FUNCTION_BLOCK ABSTRACT FB_AxisBase EXTENDS FB_ComponentBase IMPLEMENTS ITF_AxisBase
VAR CONSTANT
	//Constant declarations
	AXIS_BASE_ALARM_COUNT	: UDINT := 16;
END_VAR

VAR
	//ITF_AxisBase internal property variables
	fJogFastVelocity	: LREAL;
	fJogSlowVelocity	: LREAL;
	fTargetVelocity		: LREAL;
	
	bDriveEnabled		: BOOL;
	bInGear				: BOOL;
	bInPosition			: BOOL;
	fPosition 			: LREAL;
	fPositionSetpoint	: LREAL;
	bStopped			: BOOL;
	
	//Axis MC function blocks
	fbAxisJog: MC_Jog;
	fbAxisPower: MC_Power;
	fbAxisReset: MC_Reset;
	fbMoveAbsolute: MC_MoveAbsolute;
	fbMoveVelocity: MC_MoveVelocity;
	fbMoveRelative: MC_MoveRelative;
	fbAxisHalt: MC_Halt;
	fbAxisStop: MC_Stop;
	fbAxisHome: MC_Home;
	fbGearIn: MC_GearIn;
	fbResetDrv: FB_SoEReset;
	fbWriteParameter : MC_WriteParameter;
	
	//Alarming
	fbAxisBaseAlarms : ARRAY[1..AXIS_BASE_ALARM_COUNT] OF FB_TcAlarm;
	
	//Internal Variables
	fOverride		: LREAL := 100;		//Velocity Override
	SelectedAxis	: REFERENCE TO AXIS_REF REF= SimulationAxis;	//TODO: Make a better simulation system
	SimulationAxis: AXIS_REF;
	HardwareAxis: AXIS_REF;

	sTemp: STRING;
	stAxisBaseHMI		: ST_AxisBase_HMI;
	
	nAxisCopy: INT;
	bParamCopyComplete: BOOL;
END_VAR
VAR_IN_OUT
	MasterAxis	: AXIS_REF;
END_VAR

PROPERTY AxisRef : AXIS_REF
GET
AxisRef := SelectedAxis;
END_GET
END_PROPERTY

PROPERTY DriveEnabled : BOOL
GET
Enabled := bDriveEnabled;
END_GET
END_PROPERTY

METHOD ErrorOperation : BOOL
VAR_INPUT
END_VAR
SUPER^.ErrorOperation();

bEnabled := FALSE;
END_METHOD

METHOD GearInBasic : BOOL
VAR_IN_OUT
	master : AXIS_REF;	//Master axis to which the gearing will be made
END_VAR
IF NOT bActive THEN
	
	MasterAxis := master;		//"Master" must be specified in the FB call, so this particular variable is declared in the main FB and assigned from here
	fbGearIn.Execute := TRUE;
	
END_IF
END_METHOD

METHOD HardwareUpdate : BOOL
VAR_INPUT
END_VAR
SUPER^.HardwareUpdate();
	
//Resets the axis Drive Hardware when commanded by a "ResetDrive" Method call
fbResetDrv(
	NetId:= '', 
	Timeout:= T#10S, 
	Axis:= HardwareAxis);
	
fbResetDrv.Execute := FALSE;
END_METHOD

METHOD HMICommunication : BOOL
//Extend this method in extended FBs to communicate specific implementation data
SUPER^.HMICommunication();

//Process HMI requests
IF stAxisBaseHMI.bIncomingHMIRequest AND NOT stAxisBaseHMI.bHMICommandConfirmation THEN		//If a request has been issued by the HMI, and a previous request has not just finished being processed
	IF stAxisBaseHMI.bHMIControlAvailable THEN		//If the current conditions permit HMI control (Should be determined by the extended application components)
		IF stAxisBaseHMI.bDriveEnableHMIRequest THEN
			bEnabled := TRUE;
			stAxisBaseHMI.bHMICommandConfirmation := TRUE;	//Confirm that the request has been processed
		END_IF
		IF stAxisBaseHMI.bDriveDisableHMIRequest THEN
			bEnabled := FALSE;
			stAxisBaseHMI.bHMICommandConfirmation := TRUE;	//Confirm that the request has been processed
		END_IF
		IF stAxisBaseHMI.bSetJogFastVelocityRequest THEN
			fJogFastVelocity := stAxisBaseHMI.fSetJogFastVelocityValue;
			stAxisBaseHMI.bHMICommandConfirmation := TRUE;	//Confirm that the request has been processed
		END_IF
		IF stAxisBaseHMI.bSetJogSlowVelocityRequest THEN
			fJogSlowVelocity := stAxisBaseHMI.fSetJogSlowVelocityValue;
			stAxisBaseHMI.bHMICommandConfirmation := TRUE;	//Confirm that the request has been processed
		END_IF
		IF stAxisBaseHMI.bSetTargetVelocityRequest THEN
			fTargetVelocity := stAxisBaseHMI.bSetTargetVelocityValue;
			stAxisBaseHMI.bHMICommandConfirmation := TRUE;	//Confirm that the request has been processed
		END_IF
	END_IF
END_IF

//Update HMI status info
stAxisBaseHMI.fJogFastVelocity := fJogFastVelocity;
stAxisBaseHMI.fJogSlowVelocity := fJogSlowVelocity;
stAxisBaseHMI.fTargetVelocity := fTargetVelocity;
stAxisBaseHMI.bDriveEnabled := bDriveEnabled;
stAxisBaseHMI.bInGear := bInGear;
stAxisBaseHMI.bInPosition := bInPosition;
stAxisBaseHMI.fPosition := fPosition;
stAxisBaseHMI.fPositionSetpoint := fPositionSetpoint;
stAxisBaseHMI.bStopped := bStopped;
END_METHOD

METHOD Home : BOOL
//This method should be overridden by the extending FB based on the specific hardware configuration
END_METHOD

PROPERTY InGear : BOOL
GET
InGear := bInGear;
END_GET
END_PROPERTY

METHOD Inhibit : BOOL
VAR_INPUT
END_VAR
fbAxisPower.Override := 0;
END_METHOD

METHOD initialize : BOOL
VAR_INPUT
END_VAR

VAR
	sTemp: STRING;
END_VAR
SUPER^.initialize();

sTemp := CONCAT(CONCAT(CONCAT('Axis ', ': '), sName), ' '); 	//Creates a utility string for alarms and other messaging that reads (example text) - "Module 10 - Main Casepacker" to be followed by the alarm or message info
//TODO: Rename Event Class to AxisBase
F_CreateAllEventsInClass(	p_aAlarms := fbAxisBaseAlarms,
							nClassSize := SIZEOF(TC_EVENTS.AxisBase),
							pInitEvent := ADR(TC_EVENTS.AxisBase.InitReferenceEvent),
							sPrefix := sTemp );
END_METHOD

PROPERTY InPosition : BOOL
GET
InPosition := bInPosition;
END_GET
END_PROPERTY

METHOD Jog : BOOL
VAR_INPUT
	direction	: BOOL;			//"TRUE" for positive jog, "FALSE" for negative jog
	fast		: BOOL;			//"TRUE" for 'fast' jog, "FALSE" for 'slow' jog (As defined by Jog(Slow/Fast)Velocity Property)
END_VAR
//If the jog is currently active, allow the method to run again to ensure that the corresponding Jog bit can remain high so the jog can continue
//Otherwise, only start a jog when the axis is not already busy
IF fbAxisJog.Busy OR NOT bActive THEN
	
	fbAxisJog.JogForward:= direction; 
	fbAxisJog.JogBackwards:= NOT direction;
	
	IF fast THEN
		fbAxisJog.Velocity := fJogFastVelocity;
	ELSE
		fbAxisJog.Velocity := fJogSlowVelocity;
	END_IF
	
END_IF
END_METHOD

PROPERTY JogFastVelocity : LREAL
GET
JogFastVelocity : fJogFastVelocity;
END_GET
SET
fJogFastVelocity := JogFastVelocity;
END_SET
END_PROPERTY

PROPERTY JogSlowVelocity : LREAL
GET
JogSlowVelocity : fJogSlowVelocity;
END_GET
SET
fJogSlowVelocity : JogSlowVelocity;
END_SET
END_PROPERTY

METHOD Monitoring : BOOL
SUPER^.Monitoring();

//Cyclically updates the "Status" values from the NC-axis to the PLC (Axis1.Status...)
SelectedAxis.ReadStatus();

//Cyclically monitor all FB "Busy" bits, as well as the axis "HasJob" bit to ensure ADS communication time does not result in a delay before the "Busy" property is accurate after calling a FB
bActive := 		SimulationAxis.Status.HasJob
				OR	fbAxisJog.Busy
				OR	fbMoveAbsolute.Busy
				OR	fbMoveVelocity.Busy
				OR	fbMoveRelative.Busy
				OR	fbAxisHalt.Busy
				OR	fbAxisStop.Busy
				OR	fbAxisHome.Busy
				OR	fbGearIn.Busy;
				

//Update all internal property variables
bDriveEnabled := fbAxisPower.Status;
bInGear	:= (SelectedAxis.NcToPlc.CoupleState = 3);	//Note that this only looks for a simple gearing arrangement where this axis is a slave and not a master to any other axis
bInPosition := SelectedAxis.Status.InTargetPosition;
fPosition := SelectedAxis.NcToPlc.ActPos;
fPositionSetpoint := SelectedAxis.NcToPlc.SetPos;
bStopped := SelectedAxis.Status.StandStill;

				
//Error monitoring and event logging

IF fbAxisJog.Error AND NOT fbAxisBaseAlarms[E_AxisBase.JogError].bRaised THEN
	bError := TRUE;
	nErrorID := E_AxisBase.JogError;
	sTemp := UDINT_TO_STRING(fbAxisJog.ErrorID);
	fbAxisBaseAlarms[E_AxisBase.JogError].ipArguments.Clear().AddString(sName).AddString(sTemp);
	fbAxisBaseAlarms[E_AxisBase.JogError].Raise(0);
ELSIF NOT fbAxisJog.Error AND fbAxisBaseAlarms[E_AxisBase.JogError].bRaised THEN
	fbAxisBaseAlarms[E_AxisBase.JogError].Clear(0,0);
END_IF


IF fbAxisPower.Error AND NOT fbAxisBaseAlarms[E_AxisBase.PowerError].bRaised THEN
	bError := TRUE;
	nErrorID := E_AxisBase.PowerError;
	sTemp := UDINT_TO_STRING(fbAxisPower.ErrorID);
	fbAxisBaseAlarms[E_AxisBase.PowerError].ipArguments.Clear().AddString(sName).AddString(sTemp);
	fbAxisBaseAlarms[E_AxisBase.PowerError].Raise(0);
ELSIF NOT fbAxisPower.Error AND fbAxisBaseAlarms[E_AxisBase.PowerError].bRaised THEN
	fbAxisBaseAlarms[E_AxisBase.PowerError].Clear(0,0);
END_IF


IF fbAxisReset.Error AND NOT fbAxisBaseAlarms[E_AxisBase.ResetError].bRaised THEN
	bError := TRUE;
	nErrorID := E_AxisBase.ResetError;
	sTemp := UDINT_TO_STRING(fbAxisReset.ErrorID);
	fbAxisBaseAlarms[E_AxisBase.ResetError].ipArguments.Clear().AddString(sName).AddString(sTemp);
	fbAxisBaseAlarms[E_AxisBase.ResetError].Raise(0);
ELSIF NOT fbAxisReset.Error AND fbAxisBaseAlarms[E_AxisBase.ResetError].bRaised THEN
	fbAxisBaseAlarms[E_AxisBase.ResetError].Clear(0,0);
END_IF


IF fbMoveAbsolute.Error AND NOT fbAxisBaseAlarms[E_AxisBase.MoveAbsoluteError].bRaised THEN
	bError := TRUE;
	nErrorID := E_AxisBase.MoveAbsoluteError;
	sTemp := UDINT_TO_STRING(fbMoveAbsolute.ErrorID);
	fbAxisBaseAlarms[E_AxisBase.MoveAbsoluteError].ipArguments.Clear().AddString(sName).AddString(sTemp);
	fbAxisBaseAlarms[E_AxisBase.MoveAbsoluteError].Raise(0);
ELSIF NOT fbMoveAbsolute.Error AND fbAxisBaseAlarms[E_AxisBase.MoveAbsoluteError].bRaised THEN
	fbAxisBaseAlarms[E_AxisBase.MoveAbsoluteError].Clear(0,0);
END_IF


IF fbMoveVelocity.Error AND NOT fbAxisBaseAlarms[E_AxisBase.MoveVelocityError].bRaised THEN
	bError := TRUE;
	nErrorID := E_AxisBase.MoveVelocityError;
	sTemp := UDINT_TO_STRING(fbMoveVelocity.ErrorID);
	fbAxisBaseAlarms[E_AxisBase.MoveVelocityError].ipArguments.Clear().AddString(sName).AddString(sTemp);
	fbAxisBaseAlarms[E_AxisBase.MoveVelocityError].Raise(0);
ELSIF NOT fbMoveVelocity.Error AND fbAxisBaseAlarms[E_AxisBase.MoveVelocityError].bRaised THEN
	fbAxisBaseAlarms[E_AxisBase.MoveVelocityError].Clear(0,0);
END_IF


IF fbMoveRelative.Error AND NOT fbAxisBaseAlarms[E_AxisBase.MoveRelativeError].bRaised THEN
	bError := TRUE;
	nErrorID := E_AxisBase.MoveRelativeError;
	sTemp := UDINT_TO_STRING(fbMoveRelative.ErrorID);
	fbAxisBaseAlarms[E_AxisBase.MoveRelativeError].ipArguments.Clear().AddString(sName).AddString(sTemp);
	fbAxisBaseAlarms[E_AxisBase.MoveRelativeError].Raise(0);
ELSIF NOT fbMoveRelative.Error AND fbAxisBaseAlarms[E_AxisBase.MoveRelativeError].bRaised THEN
	fbAxisBaseAlarms[E_AxisBase.MoveRelativeError].Clear(0,0);
END_IF


IF fbAxisHalt.Error AND NOT fbAxisBaseAlarms[E_AxisBase.HaltError].bRaised THEN
	bError := TRUE;
	nErrorID := E_AxisBase.HaltError;
	sTemp := UDINT_TO_STRING(fbAxisHalt.ErrorID);
	fbAxisBaseAlarms[E_AxisBase.HaltError].ipArguments.Clear().AddString(sName).AddString(sTemp);
	fbAxisBaseAlarms[E_AxisBase.HaltError].Raise(0);
ELSIF NOT fbAxisHalt.Error AND fbAxisBaseAlarms[E_AxisBase.HaltError].bRaised THEN
	fbAxisBaseAlarms[E_AxisBase.HaltError].Clear(0,0);
END_IF


IF fbAxisStop.Error AND NOT fbAxisBaseAlarms[E_AxisBase.StopError].bRaised THEN
	bError := TRUE;
	nErrorID := E_AxisBase.StopError;
	sTemp := UDINT_TO_STRING(fbAxisStop.ErrorID);
	fbAxisBaseAlarms[E_AxisBase.StopError].ipArguments.Clear().AddString(sName).AddString(sTemp);
	fbAxisBaseAlarms[E_AxisBase.StopError].Raise(0);
ELSIF NOT fbAxisStop.Error AND fbAxisBaseAlarms[E_AxisBase.StopError].bRaised THEN
	fbAxisBaseAlarms[E_AxisBase.StopError].Clear(0,0);
END_IF


IF fbAxisHome.Error AND NOT fbAxisBaseAlarms[E_AxisBase.HomeError].bRaised THEN
	bError := TRUE;
	nErrorID := E_AxisBase.HomeError;
	sTemp := UDINT_TO_STRING(fbAxisHome.ErrorID);
	fbAxisBaseAlarms[E_AxisBase.HomeError].ipArguments.Clear().AddString(sName).AddString(sTemp);
	fbAxisBaseAlarms[E_AxisBase.HomeError].Raise(0);
ELSIF NOT fbAxisHome.Error AND fbAxisBaseAlarms[E_AxisBase.HomeError].bRaised THEN
	fbAxisBaseAlarms[E_AxisBase.HomeError].Clear(0,0);
END_IF


IF fbGearIn.Error AND NOT fbAxisBaseAlarms[E_AxisBase.GearInError].bRaised THEN
	bError := TRUE;
	nErrorID := E_AxisBase.GearInError;
	sTemp := UDINT_TO_STRING(fbGearIn.ErrorID);
	fbAxisBaseAlarms[E_AxisBase.GearInError].ipArguments.Clear().AddString(sName).AddString(sTemp);
	fbAxisBaseAlarms[E_AxisBase.GearInError].Raise(0);
ELSIF NOT fbGearIn.Error AND fbAxisBaseAlarms[E_AxisBase.GearInError].bRaised THEN
	fbAxisBaseAlarms[E_AxisBase.GearInError].Clear(0,0);
END_IF


IF fbResetDrv.Error AND NOT fbAxisBaseAlarms[E_AxisBase.ResetError].bRaised THEN
	bError := TRUE;
	nErrorID := E_AxisBase.ResetError;
	sTemp := UDINT_TO_STRING(fbResetDrv.AdsErrId);
	fbAxisBaseAlarms[E_AxisBase.ResetError].ipArguments.Clear().AddString(sName).AddString(sTemp);
	fbAxisBaseAlarms[E_AxisBase.ResetError].Raise(0);
ELSIF NOT fbResetDrv.Error AND fbAxisBaseAlarms[E_AxisBase.ResetError].bRaised THEN
	fbAxisBaseAlarms[E_AxisBase.ResetError].Clear(0,0);
END_IF

IF fbAxisPower.Override = 0 AND bActive AND NOT fbAxisBaseAlarms[E_AxisBase.CommandWhileInhibited].bRaised THEN
	bError := TRUE;
	nErrorID := E_AxisBase.CommandWhileInhibited;
	fbAxisBaseAlarms[E_AxisBase.CommandWhileInhibited].Raise(0);
ELSIF fbAxisPower.Override <> 0 AND fbAxisBaseAlarms[E_AxisBase.CommandWhileInhibited].bRaised THEN
	fbAxisBaseAlarms[E_AxisBase.CommandWhileInhibited].Clear(0,0);
END_IF

IF SimulationAxis.Status.Error AND NOT fbAxisBaseAlarms[E_AxisBase.DriveError].bRaised THEN
	bError := TRUE;
	nErrorID := E_AxisBase.DriveError;
	sTemp := UDINT_TO_STRING(SimulationAxis.Status.ErrorID);
	fbAxisBaseAlarms[E_AxisBase.DriveError].ipArguments.Clear().AddString(sName).AddString(sTemp);
	fbAxisBaseAlarms[E_AxisBase.DriveError].Raise(0);
END_IF
END_METHOD

METHOD MotionControl : BOOL
VAR_INPUT
END_VAR
//Enables the Axis for movement when commanded by an "Enable" Method call
fbAxisPower(
	Axis:= SelectedAxis,
	Enable:= bEnabled AND (bParamCopyComplete OR NOT bSimulate),
	Enable_Positive:= TRUE, 
	Enable_Negative:= TRUE, 
	Override:= fOverride, 
	BufferMode:= MC_BufferMode.MC_Aborting);


//Cyclically calls all motion fbs so that they can properly communicate to the NC
//Trigger bits (usually "Execute") are set false after each block so that external setting of execute will be read and then cleared without requiring external monitoring

//Moves the Axis to a Set Position when commanded by a "MovePosition" Method call
fbMoveAbsolute(
	Axis:= SelectedAxis,
	Velocity:= fTargetVelocity, 
	BufferMode:= MC_BufferMode.MC_Aborting );
	
fbMoveAbsolute.Execute := FALSE;

//Moves the Axis a Set Distance from its current position when commanded by a "MoveRelative" Method call
fbMoveRelative(
	Axis:= SelectedAxis, 
	Velocity:= fTargetVelocity, 
	BufferMode:= MC_BufferMode.MC_Aborting );

fbMoveRelative.Execute := FALSE;

//Starts a continuous move at a set velocity when commanded by a "MoveVelocity" Method call
fbMoveVelocity(
	Axis:= SelectedAxis, 
	Direction:= MC_Direction.MC_Positive_Direction, 
	BufferMode:= MC_BufferMode.MC_Aborting );	

fbMoveVelocity.Execute := FALSE;

//Performs a simple "Gearing" of the axis to a specified master axis at 1:1 ratio
fbGearIn(
	Master:= MasterAxis, 
	Slave:= SelectedAxis, 
	RatioNumerator:= 1, 
	RatioDenominator:= 1);
	
fbGearIn.Execute := FALSE;

//Halts the axis without disabling future commands when commanded by the "Stop" Method call
fbAxisHalt(
	Axis:= SelectedAxis,  
	BufferMode:= MC_BufferMode.MC_Aborting );	
	
fbAxisHalt.Execute := FALSE;

//Jogs the axis in a specified direction and velocity when commanded by a "Jog" Method call
fbAxisJog(
	Axis:= SelectedAxis,  
	Mode:= E_JogMode.MC_JOGMODE_CONTINOUS);

fbAxisJog.JogForward := FALSE;		//While the Jog FB does require a constant input in Continuous mode, the Method code will happen between here and the fb being called again, so the FB will not see this blip to false
fbAxisJog.JogBackwards := FALSE;	//When the "Jog" method is no longer being called, this will ensure that the jog stops on the next program cycle

//Resets the NC software axis when commanded by a "Reset" Method call
fbAxisReset(
	Axis:= SelectedAxis);

fbAxisReset.Execute := FALSE;
END_METHOD

METHOD MovePosition : BOOL
VAR_INPUT
	override 	: BOOL := FALSE;		//Allows this instruction to override another ongoing operation(This parameter is initialized so that once default parameter value functionality is added to TwinCAT, this input will not need to be set explicitly in the Method call)
	position	: LREAL;				//Desired position to which the axis should move
END_VAR
IF override OR NOT bActive THEN
	
	fbMoveAbsolute.Position := position;
	fbMoveAbsolute.Execute := TRUE;
	
END_IF
END_METHOD

METHOD MoveRelative : BOOL
VAR_INPUT
	override 	: BOOL := FALSE;		//Allows this instruction to override another ongoing operation(This parameter is initialized so that once default parameter value functionality is added to TwinCAT, this input will not need to be set explicitly in the Method call)
	distance 	: LREAL;				//Desired distance to be moved
END_VAR
IF override OR NOT bActive THEN
	
	fbMoveRelative.Distance := distance;
	fbMoveRelative.Execute := TRUE;
	
END_IF
END_METHOD

METHOD MoveVelocity : BOOL
VAR_INPUT
	override	: BOOL := FALSE;				//Allows this instruction to override another ongoing operation(This parameter is initialized so that once default parameter value functionality is added to TwinCAT, this input will not need to be set explicitly in the Method call)
	velocity	: LREAL := fTargetVelocity;		//Desired velocity for the axis (This parameter is initialized so that once default parameter value functionality is added to TwinCAT, this input will not need to be set explicitly in the Method call)
END_VAR
IF override OR NOT bActive THEN
	
	fbMoveVelocity.Velocity := velocity;
	fbMoveVelocity.Execute := TRUE;
	
END_IF
END_METHOD

PROPERTY Position : LREAL
GET
Position := fPosition;
END_GET
END_PROPERTY

PROPERTY PositionSetpoint : LREAL
GET
PositionSetpoint := fPositionSetpoint;
END_GET
END_PROPERTY

METHOD Reset : BOOL
SUPER^.Reset();

fbAxisReset.Execute := TRUE;
fbResetDrv.Execute := TRUE;
END_METHOD

METHOD ResetDrive : BOOL
fbResetDrv.Execute := FALSE;
END_METHOD

PROPERTY Simulate : BOOL
GET
END_GET
SET
END_SET
END_PROPERTY

METHOD SimulateOperation : BOOL
VAR_INPUT
END_VAR
VAR_INST
	fbWriteParam: ARRAY[1..8] OF MC_WriteParameter;
	fbAxisParamRead : ARRAY[1..8] OF MC_ReadParameter;
	fTestValue: LREAL;
	fbSetSimulationPosition: MC_SetPosition;
END_VAR
VAR
	i: INT;
END_VAR
// the need is to insure that the simulation axis always has the same dynamics and speed setpoints as the hardware axis
//copy sequence using MC2 Function Blocks

CASE nAxisCopy OF
	0:	// hold state waiting to start
		FOR i := 1 TO 8 DO
			fbAxisParamRead[i](
				Axis:= HardwareAxis,
				Enable := FALSE);
			fbWriteParam[i](
				Axis:=SimulationAxis , 
				Execute:= FALSE);
		END_FOR
		
		nAxisCopy := 10;
	10:	//read axis param
		bParamCopyComplete := FALSE;
		fbAxisParamRead[1](
			Axis:= HardwareAxis, 
			Enable:=TRUE , 
			ParameterNumber:= MC_AxisParameter.AxisMaxVelocity, 
			ReadMode:= 1, 
				Value=> fTestValue );
		fbAxisParamRead[2](
			Axis:= HardwareAxis, 
			Enable:=TRUE , 
			ParameterNumber:= MC_AxisParameter.AxisAcc, 
			ReadMode:= 1 );
		fbAxisParamRead[3](
			Axis:= HardwareAxis, 
			Enable:=TRUE , 
			ParameterNumber:= MC_AxisParameter.AxisDec, 
			ReadMode:= 1 );
		fbAxisParamRead[4](
			Axis:= HardwareAxis, 
			Enable:=TRUE , 
			ParameterNumber:= MC_AxisParameter.AxisJerk, 
			ReadMode:= 1 );
		fbAxisParamRead[5](
			Axis:= HardwareAxis, 
			Enable:=TRUE , 
			ParameterNumber:= MC_AxisParameter.AxisMaxVelocity, 
			ReadMode:= 1 );
		fbAxisParamRead[6](
			Axis:= HardwareAxis, 
			Enable:=TRUE , 
			ParameterNumber:= MC_AxisParameter.AxisManualVelocityFast, 
			ReadMode:= 1 );
		fbAxisParamRead[7](
			Axis:= HardwareAxis, 
			Enable:=TRUE , 
			ParameterNumber:= MC_AxisParameter.AxisManualVelocitySlow, 
			ReadMode:= 1 );
		fbAxisParamRead[8](
			Axis:= HardwareAxis, 
			Enable:=TRUE , 
			ParameterNumber:= MC_AxisParameter.AxisEncoderModuloValue, 
			ReadMode:= 1 );			
		IF NOT (fbAxisParamRead[1].Busy AND fbAxisParamRead[1].Valid) AND NOT 
				(fbAxisParamRead[2].Busy AND fbAxisParamRead[2].Valid) AND NOT 
				(fbAxisParamRead[3].Busy AND fbAxisParamRead[3].Valid) AND NOT 
				(fbAxisParamRead[4].Busy AND fbAxisParamRead[4].Valid) AND NOT 
				(fbAxisParamRead[5].Busy AND fbAxisParamRead[5].Valid) AND NOT 
				(fbAxisParamRead[6].Busy AND fbAxisParamRead[6].Valid) AND NOT 
				(fbAxisParamRead[7].Busy AND fbAxisParamRead[7].Valid) AND NOT 
				(fbAxisParamRead[8].Busy AND fbAxisParamRead[8].Valid)	THEN
			nAxisCopy := 20;
		ELSIF fbAxisParamRead[1].Error OR fbAxisParamRead[2].Error OR fbAxisParamRead[3].Error OR fbAxisParamRead[4].Error OR fbAxisParamRead[5].Error OR fbAxisParamRead[6].Error OR fbAxisParamRead[7].Error OR fbAxisParamRead[8].Error THEN
			nAxisCopy := 40;
		END_IF
	20:	//write axis param
		fbWriteParam[1](
			Axis:=SimulationAxis , 
			Execute:= TRUE, 
			ParameterNumber:= MC_AxisParameter.AxisVeloMax, 
			Value:= fTestValue );
		fbWriteParam[2](
			Axis:=SimulationAxis , 
			Execute:= TRUE, 
			ParameterNumber:=  MC_AxisParameter.AxisAcc, 
			Value:=fbAxisParamRead[2].Value );
		fbWriteParam[3](
			Axis:=SimulationAxis , 
			Execute:= TRUE, 
			ParameterNumber:=  MC_AxisParameter.AxisDec, 
			Value:=fbAxisParamRead[3].Value );
		fbWriteParam[4](
			Axis:=SimulationAxis , 
			Execute:= TRUE, 
			ParameterNumber:= MC_AxisParameter.AxisJerk, 
			Value:=fbAxisParamRead[4].Value );
		fbWriteParam[5](
			Axis:=SimulationAxis , 
			Execute:= TRUE, 
			ParameterNumber:= MC_AxisParameter.AxisMaxVelocity, 
			Value:=fbAxisParamRead[5].Value );
		fbWriteParam[6](
			Axis:=SimulationAxis , 
			Execute:= TRUE, 
			ParameterNumber:= MC_AxisParameter.AxisManualVelocityFast, 
			Value:=fbAxisParamRead[6].Value );
		fbWriteParam[7](
			Axis:=SimulationAxis , 
			Execute:= TRUE, 
			ParameterNumber:= MC_AxisParameter.AxisManualVelocitySlow, 
			Value:=fbAxisParamRead[7].Value );
		fbWriteParam[8](
			Axis:=SimulationAxis , 
			Execute:= TRUE, 
			ParameterNumber:= MC_AxisParameter.AxisEncoderModuloValue, 
			Value:=fbAxisParamRead[8].Value );		
		IF 	fbWriteParam[1].Done AND fbWriteParam[2].Done AND fbWriteParam[3].Done AND fbWriteParam[4].Done AND fbWriteParam[5].Done AND fbWriteParam[6].Done AND fbWriteParam[7].Done AND fbWriteParam[8].Done THEN 
			bParamCopyComplete := TRUE;
			nAxisCopy := 25;
		ELSIF fbWriteParam[1].Error OR fbWriteParam[2].Error OR fbWriteParam[3].Error OR fbWriteParam[4].Error OR fbWriteParam[5].Error OR fbWriteParam[6].Error OR fbWriteParam[7].Error OR fbWriteParam[8].Error THEN
			nAxisCopy := 40;		
		END_IF
	25: // write the hardware axis position to the simulation axis		
		fbSetSimulationPosition(
								Axis:=SimulationAxis , 
								Execute:= TRUE, 
								Position:= HardwareAxis.NcToPlc.ActPos);
		IF fbSetSimulationPosition.Done THEN 
			nAxisCopy:= 30;
		ELSIF 	fbSetSimulationPosition.Error THEN
			nAxisCopy := 40;
		END_IF
	
	30: //set selected axis
		SelectedAxis REF= SimulationAxis;
		MotionControl();
	40: //reset FB's execute and retry
		nAxisCopy :=0;
END_CASE

//SelectedAxis REF= SimulationAxis;
//MotionControl();
END_METHOD

METHOD StandardOperation : BOOL
VAR_INPUT
END_VAR
SelectedAxis REF= HardwareAxis;
nAxisCopy :=0;
MotionControl();
END_METHOD

METHOD Stop : BOOL
fbAxisHalt.Execute := TRUE;
END_METHOD

PROPERTY Stopped : BOOL
GET
Stopped := bStopped;//Axis1.Status.StandStill;
END_GET
END_PROPERTY

PROPERTY TargetVelocity : LREAL
GET
TargetVelocity : fTargetVelocity;
END_GET
SET
fTargetVelocity : TargetVelocity;
END_SET
END_PROPERTY

METHOD Uninhibit : BOOL
VAR_INPUT
END_VAR
fOverride := 100;
END_METHOD

END_FUNCTION_BLOCK

(* stored: Version 1.1.0.1, ProductVersion 3.1.4024.9
   POU FB_AxisBase: Id {2724bcaf-4a66-48a7-9f8e-fdbdfe17eb8e}, SpecialFunc None
   Folder 01_SUPER_Overrides: Id {70b354cc-2cb1-4c5f-a445-dbcd21756825}
   Folder 01_Properties: Id {f7aacb95-7ede-4f74-9420-049f48b3a795}
   Folder 02_Methods: Id {5b2faab9-1eb0-494c-97f9-6ea5d35664e2}
   Folder 02_ITF_AxisBase: Id {c94cb006-fcd3-439c-ab42-ffdbc1c4b486}
   Folder 01_Properties: Id {622640d9-38c8-4c61-88fe-751bac9bc194}
   Folder 01_Config: Id {18846eb0-bc68-4a01-94f2-7e20950c6609}
   Folder 02_Control: Id {7d88d5d2-42e2-4442-9aa3-aea79db91cb6}
   Folder 03_Status: Id {39a57548-1cdb-4874-bcf4-b3849537dccb}
   Folder 02_Methods: Id {8631449c-e13c-4da9-806d-359d178766b3}
   Folder Methods: Id {6091336e-f7a5-49a6-b5ea-b3aa6c2147ea}
   Property AxisRef: Id {e105390b-60e0-4f3f-87d6-2543e978e7e0}
   Get Get: Id {38d469f4-c2fd-48d2-818c-a001a88aa3c1}
   Property DriveEnabled: Id {c7f1ee17-db34-4e43-a694-91ab73ce00fc}
   Get Get: Id {b47da978-5009-44fe-a777-97158ddd8c0e}
   Method ErrorOperation: Id {804f7b33-db27-4ed2-8349-83fd3f9cde0f}
   Method GearInBasic: Id {d1ebe505-2ed2-4ed9-b8e9-def13444c752}
   Method HardwareUpdate: Id {aebd262c-3881-4b7c-9be9-4d42d90ff7a6}
   Method HMICommunication: Id {b0da125e-e37b-45b7-b3c0-8508142352fd}
   Method Home: Id {499c81b6-049f-44ed-a75e-5d80c1d06e89}
   Property InGear: Id {e485ac09-fe9a-4b6d-a94f-72d5ceacfd4e}
   Get Get: Id {8bb13dfc-0add-46bd-bfa6-8b0f014cd00d}
   Method Inhibit: Id {9b006364-dcbe-466d-85f5-56fbd40c1fa5}
   Method initialize: Id {5fde8ae3-1f58-43c0-8ce3-aad5840cbb70}
   Property InPosition: Id {de0a94d7-5134-4915-8d09-8bde4bf62b71}
   Get Get: Id {8040b295-8ac3-4387-a918-4d660c3a66dc}
   Method Jog: Id {7f8f32e3-9f32-4eeb-b744-6da4e93681ab}
   Property JogFastVelocity: Id {373ad61c-a187-45f5-967f-0ac675c75f31}
   Get Get: Id {8361121e-bedc-4874-acd3-a6261146f5d2}
   Set Set: Id {e489f0ad-8f0e-4429-b255-4423642cdc1a}
   Property JogSlowVelocity: Id {1c4b0209-b9c2-4dd5-a975-ae2265c3e153}
   Get Get: Id {a778afc0-afe5-4e65-b514-1edb0437b76b}
   Set Set: Id {320a0644-77d6-4836-8f13-12e9c54aea00}
   Method Monitoring: Id {bb6fc4ed-d443-4e5b-b9ab-eb66e37cd61b}
   Method MotionControl: Id {24aa628f-77c9-4939-b88a-d6572a4e5a53}
   Method MovePosition: Id {4457c8ba-d59c-46c6-a0cb-8d5fd534908c}
   Method MoveRelative: Id {736eb44c-6c1e-4102-b9d5-d6446b49d731}
   Method MoveVelocity: Id {fe47d529-d067-4610-afa7-028a0d8a9831}
   Property Position: Id {735f7abc-47fb-4467-aae1-b71e86502f6b}
   Get Get: Id {b21971e3-905e-489e-9dc2-aa78d1607290}
   Property PositionSetpoint: Id {98e0caf3-a5ce-473c-a05f-9d2a5acf3ce1}
   Get Get: Id {a7e12c4c-7147-45b1-b3bb-f343af67c769}
   Method Reset: Id {54a459a8-7f40-4053-bdb8-feea4d756ed7}
   Method ResetDrive: Id {61a188ee-6e1c-4070-8317-83a705f013d8}
   Property Simulate: Id {0efad7c3-dfea-405c-94fb-a00cc1a2a266}
   Get Get: Id {b8f83469-562b-4225-a7d1-ccd4df07420a}
   Set Set: Id {34f3db18-fa78-4adc-b908-d8398e3253ee}
   Method SimulateOperation: Id {d1ff29c4-9c3d-4f08-b25b-d926ccfd1f38}
   Method StandardOperation: Id {41f73aab-0313-4f40-bdbc-bd3027fb897e}
   Method Stop: Id {34368b61-2529-4fbb-9bd5-94608a09587b}
   Property Stopped: Id {e5d267d6-da40-4494-bed4-1f6fbd96137d}
   Get Get: Id {9d0759f2-a208-47e4-a3e0-4201ee14c7f8}
   Property TargetVelocity: Id {74cf7284-2549-4bf5-b6ee-5e705534f1be}
   Get Get: Id {8b10f2d5-2236-4ab3-9318-4840e60faf8c}
   Set Set: Id {78fcc4c5-e7f9-4e26-ba73-aac4631ae881}
   Method Uninhibit: Id {5eff14cf-20b3-463c-b066-34b02f88809f} *)
